// TIA Portal V21 export
DATA_BLOCK "Simulation_DB"   // DB2
{ S7_Optimized_Access := 'TRUE'; DB_Accessible_From_OPC_UA := 'FALSE' }
// stored: AutoNumber false, DBAccessibleFromOPCUA false, DBAccessibleFromWebserver false, MemoryReserve 100
   VAR
      Simulation { ExternalAccessible := 'False'; ExternalVisible := 'False'; ExternalWritable := 'False'} : Bool;
      DigitalInputs : Struct
         EmergencyStop : Bool;
         Start : Bool;
         Stop : Bool;
         Reset : Bool;
         ContactorON : Array[1..2] of Bool;
         SoftstartON : Array[1..2] of Bool;
         SoftstartBypassed : Array[1..2] of Bool;
         SoftstartFault : Array[1..2] of Bool;
         Protection : Array[1..2] of Bool;
      END_STRUCT;
      TankLevel { ExternalWritable := 'False'} : Array[1..2] of Int;
   END_VAR
BEGIN
END_DATA_BLOCK
